// TIA Portal project "SERVO_2_AXIS" (V15.1)

(* hardware
DEVICE "S7-1200 station_1"  S7-1200 Station
   slot 0: "Rack_0"  S7-1200 Rack  Rack  V1.0
   slot 1: "PLC_1"  CPU 1214C DC/DC/DC  6ES7 214-1AG40-0XB0  V4.2
DEVICE "PC-System_1"  SIMATIC PC station
   slot 0: "SIMATIC PC station"  Rail  SIMATIC PC-Station  V1.0
      slot 125: "Stationmanager"  Station_Manager  V6.0.4
   slot 1: "HMI_RT_1"  WinCC RT Advanced  6AV2 104-0xxxx-xxxx  15.1.0.0
      slot 33792: "Host interface"  Host interface
   slot 2: "IE general_1"  IE General  IE_CP  V8.2.0
*)

// ===== PLC "PLC_1"  CPU 1214C DC/DC/DC =====

VAR_GLOBAL   // PLC tag table "Default tag table"
   "Axis_X_Pulse" AT %Q0.0 : Bool;
   "Axis_X_Direction" AT %Q0.1 : Bool;
   "Axis_Y_Pulse" AT %Q0.2 : Bool;
   "Axis_Y_Direction" AT %Q0.3 : Bool;
   "Tag_1" AT %M40.0 : Bool;
   "Set_Home_X" AT %M40.1 : Bool;
   "Thuận _X" AT %M40.2 : Bool;
   "Ngược_X" AT %M40.3 : Bool;
   "Speed_X" AT %MD10 : Real;
   "Enable_Y" AT %M50.0 : Bool;
   "Set_Home_Y" AT %M50.1 : Bool;
   "Thuận_Y" AT %M50.2 : Bool;
   "Ngược_Y" AT %M50.3 : Bool;
   "Speed_Y" AT %MD20 : Real;
   "Location_To_X" AT %MD14 : Real;
   "Start_X" AT %M40.4 : Bool;
   "Start_Y" AT %M50.4 : Bool;
   "Location_To_Y" AT %MD24 : Real;
   "Save_Location_X1" AT %M40.5 : Bool;
   "Save_Location_X2" AT %M40.6 : Bool;
   "Save_Location_X3" AT %M40.7 : Bool;
   "Save_Location_X4" AT %M41.0 : Bool;
   "Save_Location_X5" AT %M41.1 : Bool;
   "Save_Location_Y1" AT %M50.5 : Bool;
   "Save_Location_Y2" AT %M50.6 : Bool;
   "Save_Location_Y3" AT %M50.7 : Bool;
   "Save_Location_Y4" AT %M51.0 : Bool;
   "Save_Location_Y5" AT %M51.1 : Bool;
   "Input_location_X" AT %MW60 : Word;
   "Input_location_Y" AT %MW70 : Word;
   "System_Byte" AT %MB1 : Byte;
   "FirstScan" AT %M1.0 : Bool;
   "DiagStatusUpdate" AT %M1.1 : Bool;
   "AlwaysTRUE" AT %M1.2 : Bool;
   "AlwaysFALSE" AT %M1.3 : Bool;
   "X1" AT %M2.0 : Bool;
   "X2" AT %M2.1 : Bool;
   "X3" AT %M2.2 : Bool;
   "X4" AT %M2.3 : Bool;
   "X5" AT %M2.4 : Bool;
   "Y1" AT %M2.5 : Bool;
   "Y2" AT %M2.6 : Bool;
   "Y3" AT %M3.0 : Bool;
   "Y4" AT %M3.1 : Bool;
   "Y5" AT %M3.2 : Bool;
   "X1Y1" AT %M3.3 : Bool;
   "X1Y2" AT %M3.4 : Bool;
   "X1Y3" AT %M3.5 : Bool;
   "X1Y4" AT %M3.6 : Bool;
   "X1Y5" AT %M3.7 : Bool;
   "X2Y1" AT %M4.0 : Bool;
   "X2Y2" AT %M4.1 : Bool;
   "X2Y3" AT %M4.2 : Bool;
   "X2Y4" AT %M4.3 : Bool;
   "X2Y5" AT %M4.4 : Bool;
   "X3Y1" AT %M4.5 : Bool;
   "X3Y2" AT %M4.6 : Bool;
   "X3Y3" AT %M4.7 : Bool;
   "X3Y4" AT %M5.0 : Bool;
   "X3Y5" AT %M5.1 : Bool;
   "X4Y1" AT %M5.2 : Bool;
   "X4Y2" AT %M5.3 : Bool;
   "X4Y3" AT %M5.4 : Bool;
   "X4Y4" AT %M5.5 : Bool;
   "X4Y5" AT %M5.6 : Bool;
   "X5Y1" AT %M5.7 : Bool;
   "X5Y2" AT %M6.0 : Bool;
   "X5Y3" AT %M6.1 : Bool;
   "X5Y4" AT %M6.2 : Bool;
   "X5Y5" AT %M6.3 : Bool;
END_VAR

DATA_BLOCK "Location_X"   // DB3
{ S7_Optimized_Access := 'FALSE' }
VERSION : 0.1
   VAR
      Location_X : Array[1..5] of Real;
   END_VAR
BEGIN
END_DATA_BLOCK

DATA_BLOCK "Location_Y"   // DB4
{ S7_Optimized_Access := 'FALSE' }
VERSION : 0.1
   VAR
      Location_Y : Array[1..5] of Real;
   END_VAR
BEGIN
END_DATA_BLOCK

DATA_BLOCK "Axis_X"   // DB1, Motion_DB
{ S7_Optimized_Access := 'TRUE' }
AUTHOR : SIMATIC
FAMILY : BasicMC
NAME : TO_PosAx
VERSION : 6.0
// stored: InstanceOfName TO_PositioningAxis
"TO_PositioningAxis"
BEGIN
   // Axis.LengthUnitNormalized.Distance = 1013
   // Axis.DirectionOutputEnabledCU = TRUE
   // Axis.OnlinePtoModeCU = 16#0000_0002
   // Axis.SelectedChannel2EnumCU = %Q0.1
   // Axis.SelectedChannel1EnumCU = %Q0.0
   // Pulse.MinDeltaDeltaFrequencyCU = 0.004
   // Pulse.MaxDeltaDeltaFrequencyCU = 1.0E+10
   // Pulse.MinDeltaFrequencyCU = 0.005
   // Pulse.MaxDeltaFrequencyCU = 9.5E+9
   // Pulse.MinFrequencyCU = 1.0
   // Pulse.MaxFrequencyCU = 100000.0
   // Pulse.OutputSourceCU = 16#0000_0000
   // Axis.SelectPTO = 0
END_DATA_BLOCK

DATA_BLOCK "Axis_Y"   // DB2, Motion_DB
{ S7_Optimized_Access := 'TRUE' }
AUTHOR : SIMATIC
FAMILY : BasicMC
NAME : TO_PosAx
VERSION : 6.0
// stored: InstanceOfName TO_PositioningAxis
"TO_PositioningAxis"
BEGIN
   // Axis.LengthUnitNormalized.Distance = 1013
   // Axis.DirectionOutputEnabledCU = TRUE
   // Axis.OnlinePtoModeCU = 16#0000_0002
   // Axis.SelectedChannel2EnumCU = %Q0.3
   // Axis.SelectedChannel1EnumCU = %Q0.2
   // Pulse.MinDeltaDeltaFrequencyCU = 0.004
   // Pulse.MaxDeltaDeltaFrequencyCU = 1.0E+10
   // Pulse.MinDeltaFrequencyCU = 0.005
   // Pulse.MaxDeltaFrequencyCU = 9.5E+9
   // Pulse.MinFrequencyCU = 1.0
   // Pulse.MaxFrequencyCU = 100000.0
   // Pulse.OutputSourceCU = 16#0000_0000
   // Axis.SelectPTO = 1
   // Axis.OnlinePtoIndexCU = 1
END_DATA_BLOCK

FUNCTION "Power_X" : Void   // FC1, LAD
{ S7_Optimized_Access := 'TRUE' }
VERSION : 0.1
BEGIN

REGION Network 1
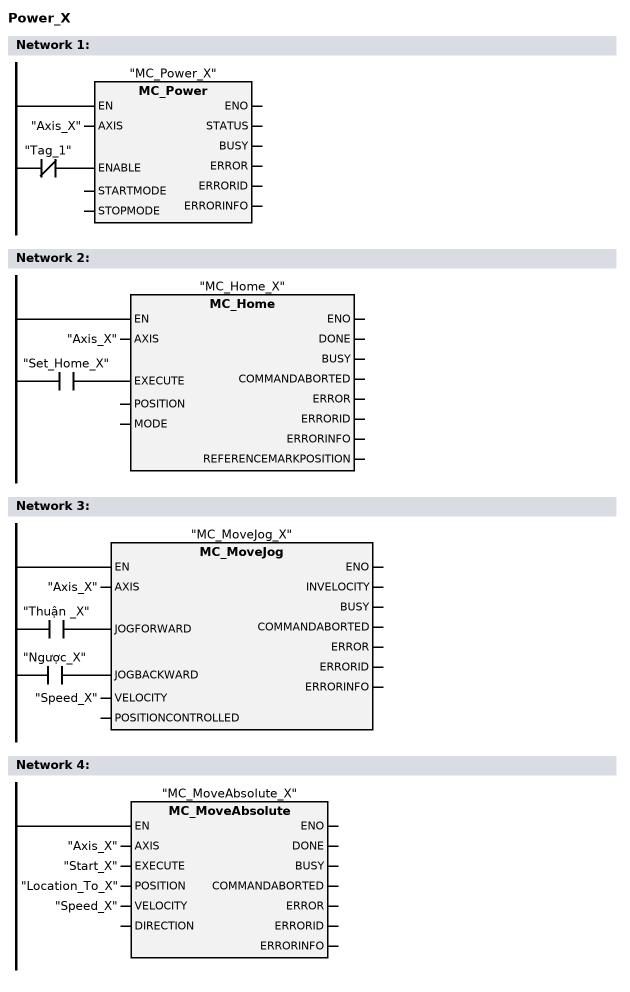
   "MC_Power_X"(Axis := "Axis_X", Enable := NOT "Tag_1");   // MC_Power
END_REGION

REGION Network 2
   "MC_Home_X"(Axis := "Axis_X", Execute := "Set_Home_X");   // MC_Home
END_REGION

REGION Network 3
   "MC_MoveJog_X"(Axis := "Axis_X", JogForward := "Thuận _X", JogBackward := "Ngược_X", Velocity := "Speed_X");   // MC_MoveJog
END_REGION

REGION Network 4
   "MC_MoveAbsolute_X"(Axis := "Axis_X",   // MC_MoveAbsolute
                       Execute := "Start_X",
                       Position := "Location_To_X",
                       Velocity := "Speed_X");
END_REGION
END_FUNCTION

FUNCTION "Power_Y" : Void   // FC2, LAD
{ S7_Optimized_Access := 'TRUE' }
VERSION : 0.1
BEGIN

REGION Network 1
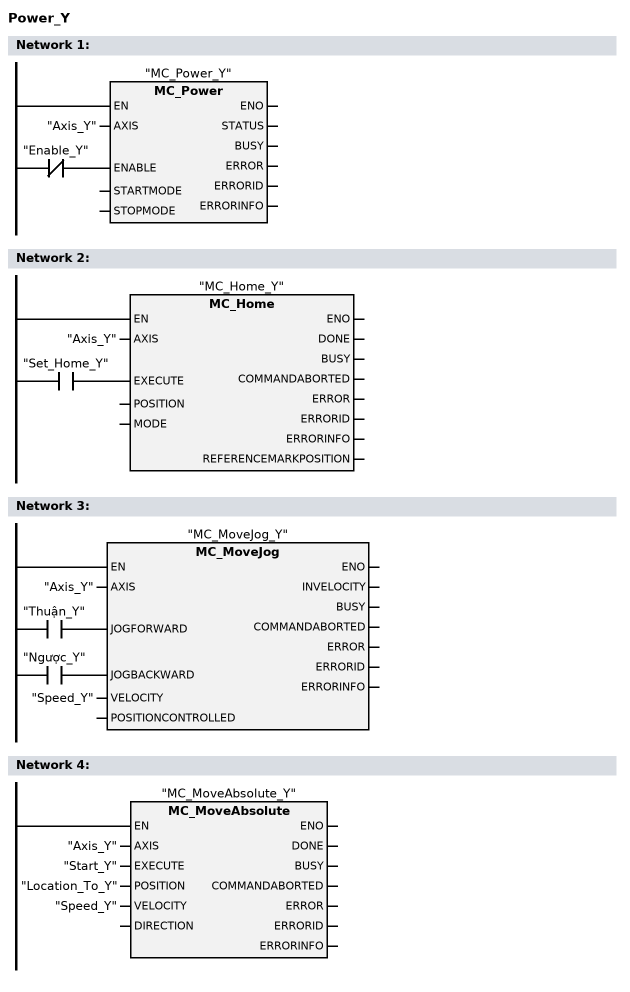
   "MC_Power_Y"(Axis := "Axis_Y", Enable := NOT "Enable_Y");   // MC_Power
END_REGION

REGION Network 2
   "MC_Home_Y"(Axis := "Axis_Y", Execute := "Set_Home_Y");   // MC_Home
END_REGION

REGION Network 3
   "MC_MoveJog_Y"(Axis := "Axis_Y", JogForward := "Thuận_Y", JogBackward := "Ngược_Y", Velocity := "Speed_Y");   // MC_MoveJog
END_REGION

REGION Network 4
   "MC_MoveAbsolute_Y"(Axis := "Axis_Y",   // MC_MoveAbsolute
                       Execute := "Start_Y",
                       Position := "Location_To_Y",
                       Velocity := "Speed_Y");
END_REGION
END_FUNCTION

FUNCTION "Save_Location_X" : Void   // FC3, LAD
{ S7_Optimized_Access := 'TRUE' }
VERSION : 0.1
BEGIN

REGION Network 1
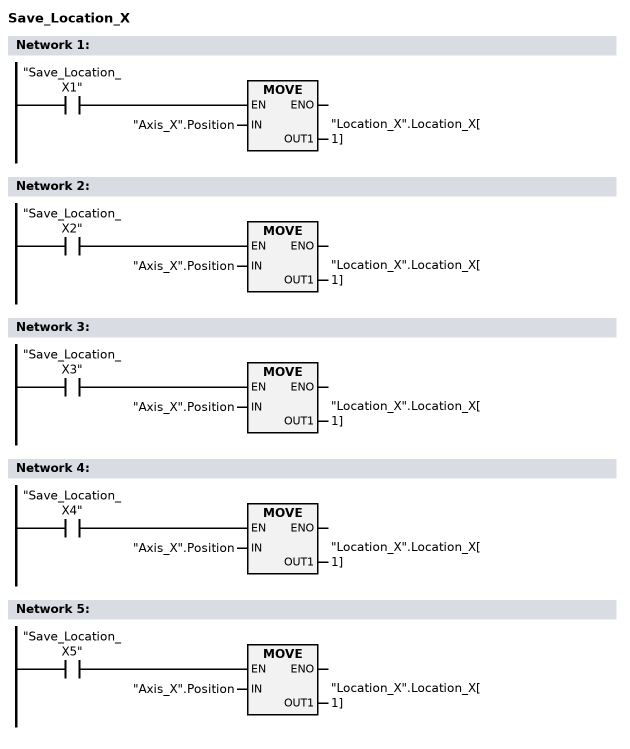
   RUNG wire#powerrail
      Contact( "Save_Location_X1" )
      Move(in := "Axis_X".Position, out1 => "Location_X".Location_X[1])
   END_RUNG
   // the same network as SCL:
   IF "Save_Location_X1" THEN "Location_X".Location_X[1] := "Axis_X".Position; END_IF;
END_REGION

REGION Network 2
   RUNG wire#powerrail
      Contact( "Save_Location_X2" )
      Move(in := "Axis_X".Position, out1 => "Location_X".Location_X[1])
   END_RUNG
   // the same network as SCL:
   IF "Save_Location_X2" THEN "Location_X".Location_X[1] := "Axis_X".Position; END_IF;
END_REGION

REGION Network 3
   RUNG wire#powerrail
      Contact( "Save_Location_X3" )
      Move(in := "Axis_X".Position, out1 => "Location_X".Location_X[1])
   END_RUNG
   // the same network as SCL:
   IF "Save_Location_X3" THEN "Location_X".Location_X[1] := "Axis_X".Position; END_IF;
END_REGION

REGION Network 4
   RUNG wire#powerrail
      Contact( "Save_Location_X4" )
      Move(in := "Axis_X".Position, out1 => "Location_X".Location_X[1])
   END_RUNG
   // the same network as SCL:
   IF "Save_Location_X4" THEN "Location_X".Location_X[1] := "Axis_X".Position; END_IF;
END_REGION

REGION Network 5
   RUNG wire#powerrail
      Contact( "Save_Location_X5" )
      Move(in := "Axis_X".Position, out1 => "Location_X".Location_X[1])
   END_RUNG
   // the same network as SCL:
   IF "Save_Location_X5" THEN "Location_X".Location_X[1] := "Axis_X".Position; END_IF;
END_REGION
END_FUNCTION

FUNCTION "Save_Location_Y" : Void   // FC4, LAD
{ S7_Optimized_Access := 'TRUE' }
VERSION : 0.1
BEGIN

REGION Network 1
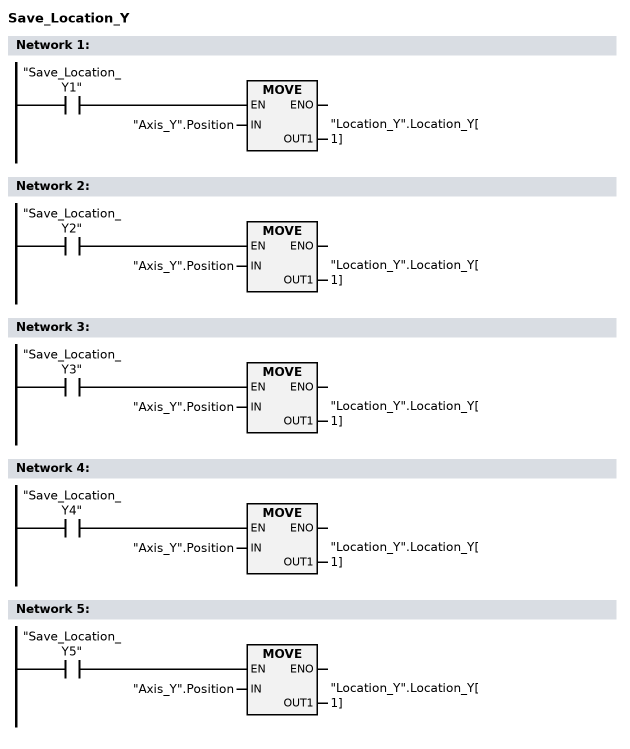
   RUNG wire#powerrail
      Contact( "Save_Location_Y1" )
      Move(in := "Axis_Y".Position, out1 => "Location_Y".Location_Y[1])
   END_RUNG
   // the same network as SCL:
   IF "Save_Location_Y1" THEN "Location_Y".Location_Y[1] := "Axis_Y".Position; END_IF;
END_REGION

REGION Network 2
   RUNG wire#powerrail
      Contact( "Save_Location_Y2" )
      Move(in := "Axis_Y".Position, out1 => "Location_Y".Location_Y[1])
   END_RUNG
   // the same network as SCL:
   IF "Save_Location_Y2" THEN "Location_Y".Location_Y[1] := "Axis_Y".Position; END_IF;
END_REGION

REGION Network 3
   RUNG wire#powerrail
      Contact( "Save_Location_Y3" )
      Move(in := "Axis_Y".Position, out1 => "Location_Y".Location_Y[1])
   END_RUNG
   // the same network as SCL:
   IF "Save_Location_Y3" THEN "Location_Y".Location_Y[1] := "Axis_Y".Position; END_IF;
END_REGION

REGION Network 4
   RUNG wire#powerrail
      Contact( "Save_Location_Y4" )
      Move(in := "Axis_Y".Position, out1 => "Location_Y".Location_Y[1])
   END_RUNG
   // the same network as SCL:
   IF "Save_Location_Y4" THEN "Location_Y".Location_Y[1] := "Axis_Y".Position; END_IF;
END_REGION

REGION Network 5
   RUNG wire#powerrail
      Contact( "Save_Location_Y5" )
      Move(in := "Axis_Y".Position, out1 => "Location_Y".Location_Y[1])
   END_RUNG
   // the same network as SCL:
   IF "Save_Location_Y5" THEN "Location_Y".Location_Y[1] := "Axis_Y".Position; END_IF;
END_REGION
END_FUNCTION

FUNCTION "Call_Location_X" : Void   // FC5, LAD
{ S7_Optimized_Access := 'TRUE' }
VERSION : 0.1
BEGIN

REGION Network 1
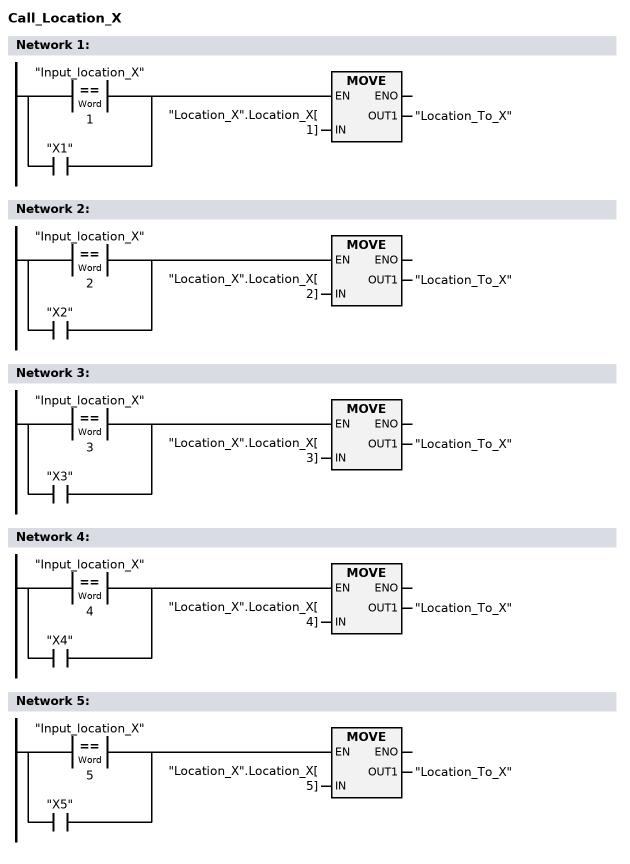
   RUNG wire#powerrail
      { S7_Templates := "SrcType := Word" } EQ_Contact(in1 := "Input_location_X", in2 := 1)
      wire#w1
      Move(in := "Location_X".Location_X[1], out1 => "Location_To_X")
   END_RUNG
   RUNG wire#powerrail
      Contact( "X1" )
   END_RUNG wire#w1
   // the same network as SCL:
   IF ("Input_location_X" = 1) OR "X1" THEN "Location_To_X" := "Location_X".Location_X[1]; END_IF;
END_REGION

REGION Network 2
   RUNG wire#powerrail
      { S7_Templates := "SrcType := Word" } EQ_Contact(in1 := "Input_location_X", in2 := 2)
      wire#w1
      Move(in := "Location_X".Location_X[2], out1 => "Location_To_X")
   END_RUNG
   RUNG wire#powerrail
      Contact( "X2" )
   END_RUNG wire#w1
   // the same network as SCL:
   IF ("Input_location_X" = 2) OR "X2" THEN "Location_To_X" := "Location_X".Location_X[2]; END_IF;
END_REGION

REGION Network 3
   RUNG wire#powerrail
      { S7_Templates := "SrcType := Word" } EQ_Contact(in1 := "Input_location_X", in2 := 3)
      wire#w1
      Move(in := "Location_X".Location_X[3], out1 => "Location_To_X")
   END_RUNG
   RUNG wire#powerrail
      Contact( "X3" )
   END_RUNG wire#w1
   // the same network as SCL:
   IF ("Input_location_X" = 3) OR "X3" THEN "Location_To_X" := "Location_X".Location_X[3]; END_IF;
END_REGION

REGION Network 4
   RUNG wire#powerrail
      { S7_Templates := "SrcType := Word" } EQ_Contact(in1 := "Input_location_X", in2 := 4)
      wire#w1
      Move(in := "Location_X".Location_X[4], out1 => "Location_To_X")
   END_RUNG
   RUNG wire#powerrail
      Contact( "X4" )
   END_RUNG wire#w1
   // the same network as SCL:
   IF ("Input_location_X" = 4) OR "X4" THEN "Location_To_X" := "Location_X".Location_X[4]; END_IF;
END_REGION

REGION Network 5
   RUNG wire#powerrail
      { S7_Templates := "SrcType := Word" } EQ_Contact(in1 := "Input_location_X", in2 := 5)
      wire#w1
      Move(in := "Location_X".Location_X[5], out1 => "Location_To_X")
   END_RUNG
   RUNG wire#powerrail
      Contact( "X5" )
   END_RUNG wire#w1
   // the same network as SCL:
   IF ("Input_location_X" = 5) OR "X5" THEN "Location_To_X" := "Location_X".Location_X[5]; END_IF;
END_REGION
END_FUNCTION

FUNCTION "Call_Location_Y" : Void   // FC6, LAD
{ S7_Optimized_Access := 'TRUE' }
VERSION : 0.1
BEGIN

REGION Network 1
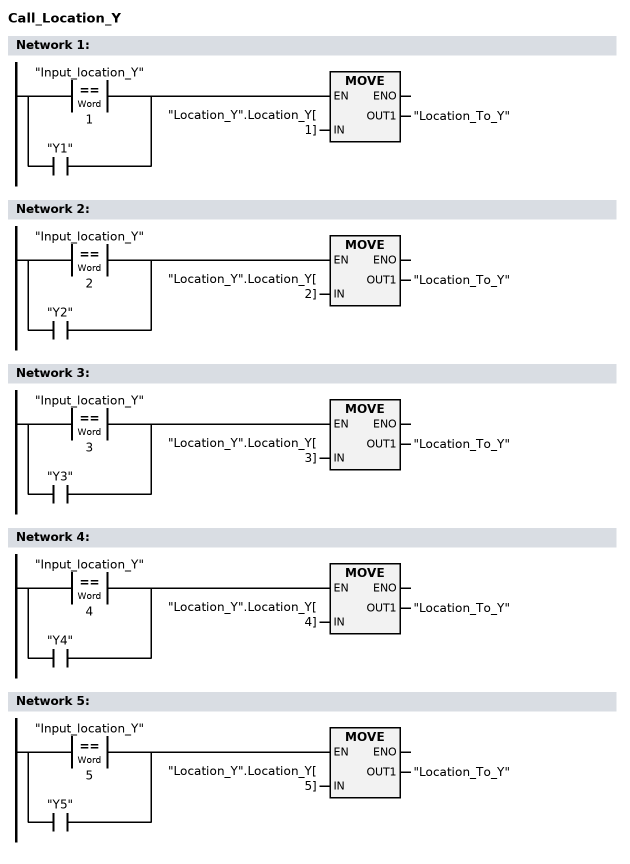
   RUNG wire#powerrail
      { S7_Templates := "SrcType := Word" } EQ_Contact(in1 := "Input_location_Y", in2 := 1)
      wire#w1
      Move(in := "Location_Y".Location_Y[1], out1 => "Location_To_Y")
   END_RUNG
   RUNG wire#powerrail
      Contact( "Y1" )
   END_RUNG wire#w1
   // the same network as SCL:
   IF ("Input_location_Y" = 1) OR "Y1" THEN "Location_To_Y" := "Location_Y".Location_Y[1]; END_IF;
END_REGION

REGION Network 2
   RUNG wire#powerrail
      { S7_Templates := "SrcType := Word" } EQ_Contact(in1 := "Input_location_Y", in2 := 2)
      wire#w1
      Move(in := "Location_Y".Location_Y[2], out1 => "Location_To_Y")
   END_RUNG
   RUNG wire#powerrail
      Contact( "Y2" )
   END_RUNG wire#w1
   // the same network as SCL:
   IF ("Input_location_Y" = 2) OR "Y2" THEN "Location_To_Y" := "Location_Y".Location_Y[2]; END_IF;
END_REGION

REGION Network 3
   RUNG wire#powerrail
      { S7_Templates := "SrcType := Word" } EQ_Contact(in1 := "Input_location_Y", in2 := 3)
      wire#w1
      Move(in := "Location_Y".Location_Y[3], out1 => "Location_To_Y")
   END_RUNG
   RUNG wire#powerrail
      Contact( "Y3" )
   END_RUNG wire#w1
   // the same network as SCL:
   IF ("Input_location_Y" = 3) OR "Y3" THEN "Location_To_Y" := "Location_Y".Location_Y[3]; END_IF;
END_REGION

REGION Network 4
   RUNG wire#powerrail
      { S7_Templates := "SrcType := Word" } EQ_Contact(in1 := "Input_location_Y", in2 := 4)
      wire#w1
      Move(in := "Location_Y".Location_Y[4], out1 => "Location_To_Y")
   END_RUNG
   RUNG wire#powerrail
      Contact( "Y4" )
   END_RUNG wire#w1
   // the same network as SCL:
   IF ("Input_location_Y" = 4) OR "Y4" THEN "Location_To_Y" := "Location_Y".Location_Y[4]; END_IF;
END_REGION

REGION Network 5
   RUNG wire#powerrail
      { S7_Templates := "SrcType := Word" } EQ_Contact(in1 := "Input_location_Y", in2 := 5)
      wire#w1
      Move(in := "Location_Y".Location_Y[5], out1 => "Location_To_Y")
   END_RUNG
   RUNG wire#powerrail
      Contact( "Y5" )
   END_RUNG wire#w1
   // the same network as SCL:
   IF ("Input_location_Y" = 5) OR "Y5" THEN "Location_To_Y" := "Location_Y".Location_Y[5]; END_IF;
END_REGION
END_FUNCTION

FUNCTION "XY" : Void   // FC7, LAD
{ S7_Optimized_Access := 'TRUE' }
VERSION : 0.1
BEGIN

REGION Network 1
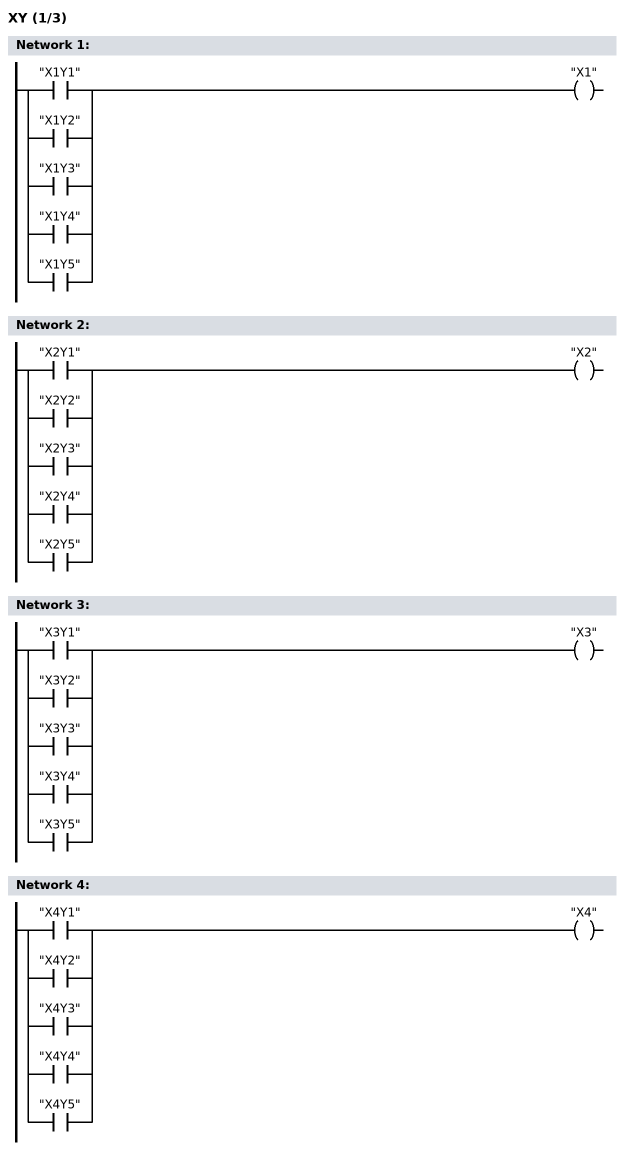
   RUNG wire#powerrail
      Contact( "X1Y1" )
      wire#w1
      Coil( "X1" )
   END_RUNG
   RUNG wire#powerrail
      Contact( "X1Y2" )
   END_RUNG wire#w1
   RUNG wire#powerrail
      Contact( "X1Y3" )
   END_RUNG wire#w1
   RUNG wire#powerrail
      Contact( "X1Y4" )
   END_RUNG wire#w1
   RUNG wire#powerrail
      Contact( "X1Y5" )
   END_RUNG wire#w1
   // the same network as SCL:
   "X1" := "X1Y1" OR "X1Y2" OR "X1Y3" OR "X1Y4" OR "X1Y5";
END_REGION

REGION Network 2
   RUNG wire#powerrail
      Contact( "X2Y1" )
      wire#w1
      Coil( "X2" )
   END_RUNG
   RUNG wire#powerrail
      Contact( "X2Y2" )
   END_RUNG wire#w1
   RUNG wire#powerrail
      Contact( "X2Y3" )
   END_RUNG wire#w1
   RUNG wire#powerrail
      Contact( "X2Y4" )
   END_RUNG wire#w1
   RUNG wire#powerrail
      Contact( "X2Y5" )
   END_RUNG wire#w1
   // the same network as SCL:
   "X2" := "X2Y1" OR "X2Y2" OR "X2Y3" OR "X2Y4" OR "X2Y5";
END_REGION

REGION Network 3
   RUNG wire#powerrail
      Contact( "X3Y1" )
      wire#w1
      Coil( "X3" )
   END_RUNG
   RUNG wire#powerrail
      Contact( "X3Y2" )
   END_RUNG wire#w1
   RUNG wire#powerrail
      Contact( "X3Y3" )
   END_RUNG wire#w1
   RUNG wire#powerrail
      Contact( "X3Y4" )
   END_RUNG wire#w1
   RUNG wire#powerrail
      Contact( "X3Y5" )
   END_RUNG wire#w1
   // the same network as SCL:
   "X3" := "X3Y1" OR "X3Y2" OR "X3Y3" OR "X3Y4" OR "X3Y5";
END_REGION

REGION Network 4
   RUNG wire#powerrail
      Contact( "X4Y1" )
      wire#w1
      Coil( "X4" )
   END_RUNG
   RUNG wire#powerrail
      Contact( "X4Y2" )
   END_RUNG wire#w1
   RUNG wire#powerrail
      Contact( "X4Y3" )
   END_RUNG wire#w1
   RUNG wire#powerrail
      Contact( "X4Y4" )
   END_RUNG wire#w1
   RUNG wire#powerrail
      Contact( "X4Y5" )
   END_RUNG wire#w1
   // the same network as SCL:
   "X4" := "X4Y1" OR "X4Y2" OR "X4Y3" OR "X4Y4" OR "X4Y5";
END_REGION

REGION Network 5
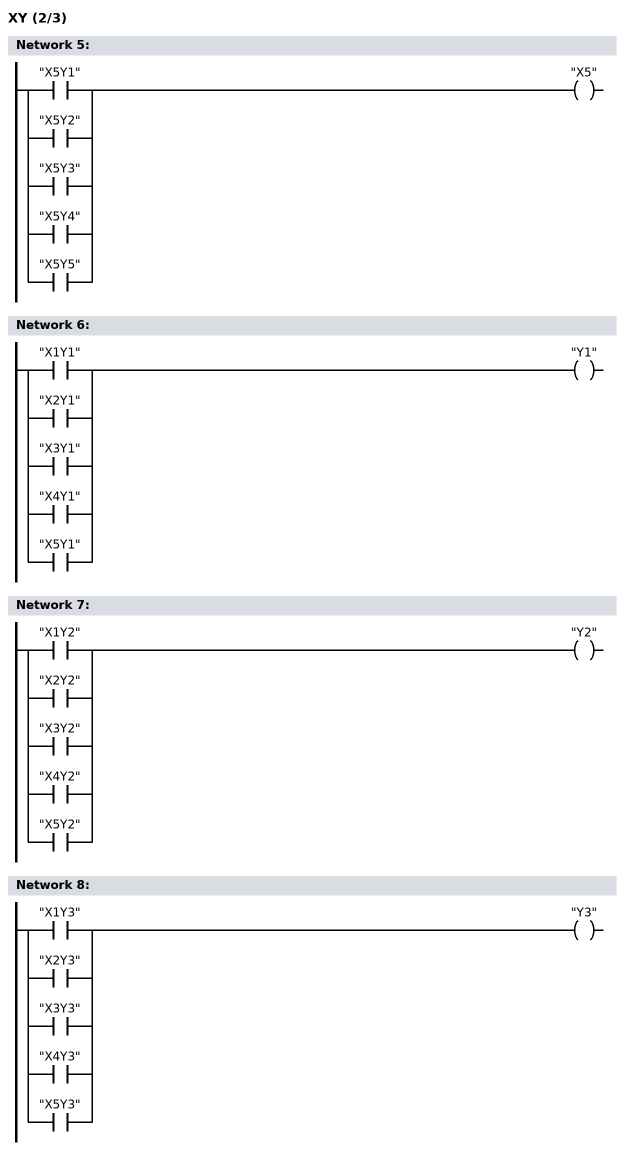
   RUNG wire#powerrail
      Contact( "X5Y1" )
      wire#w1
      Coil( "X5" )
   END_RUNG
   RUNG wire#powerrail
      Contact( "X5Y2" )
   END_RUNG wire#w1
   RUNG wire#powerrail
      Contact( "X5Y3" )
   END_RUNG wire#w1
   RUNG wire#powerrail
      Contact( "X5Y4" )
   END_RUNG wire#w1
   RUNG wire#powerrail
      Contact( "X5Y5" )
   END_RUNG wire#w1
   // the same network as SCL:
   "X5" := "X5Y1" OR "X5Y2" OR "X5Y3" OR "X5Y4" OR "X5Y5";
END_REGION

REGION Network 6
   RUNG wire#powerrail
      Contact( "X1Y1" )
      wire#w1
      Coil( "Y1" )
   END_RUNG
   RUNG wire#powerrail
      Contact( "X2Y1" )
   END_RUNG wire#w1
   RUNG wire#powerrail
      Contact( "X3Y1" )
   END_RUNG wire#w1
   RUNG wire#powerrail
      Contact( "X4Y1" )
   END_RUNG wire#w1
   RUNG wire#powerrail
      Contact( "X5Y1" )
   END_RUNG wire#w1
   // the same network as SCL:
   "Y1" := "X1Y1" OR "X2Y1" OR "X3Y1" OR "X4Y1" OR "X5Y1";
END_REGION

REGION Network 7
   RUNG wire#powerrail
      Contact( "X1Y2" )
      wire#w1
      Coil( "Y2" )
   END_RUNG
   RUNG wire#powerrail
      Contact( "X2Y2" )
   END_RUNG wire#w1
   RUNG wire#powerrail
      Contact( "X3Y2" )
   END_RUNG wire#w1
   RUNG wire#powerrail
      Contact( "X4Y2" )
   END_RUNG wire#w1
   RUNG wire#powerrail
      Contact( "X5Y2" )
   END_RUNG wire#w1
   // the same network as SCL:
   "Y2" := "X1Y2" OR "X2Y2" OR "X3Y2" OR "X4Y2" OR "X5Y2";
END_REGION

REGION Network 8
   RUNG wire#powerrail
      Contact( "X1Y3" )
      wire#w1
      Coil( "Y3" )
   END_RUNG
   RUNG wire#powerrail
      Contact( "X2Y3" )
   END_RUNG wire#w1
   RUNG wire#powerrail
      Contact( "X3Y3" )
   END_RUNG wire#w1
   RUNG wire#powerrail
      Contact( "X4Y3" )
   END_RUNG wire#w1
   RUNG wire#powerrail
      Contact( "X5Y3" )
   END_RUNG wire#w1
   // the same network as SCL:
   "Y3" := "X1Y3" OR "X2Y3" OR "X3Y3" OR "X4Y3" OR "X5Y3";
END_REGION

REGION Network 9
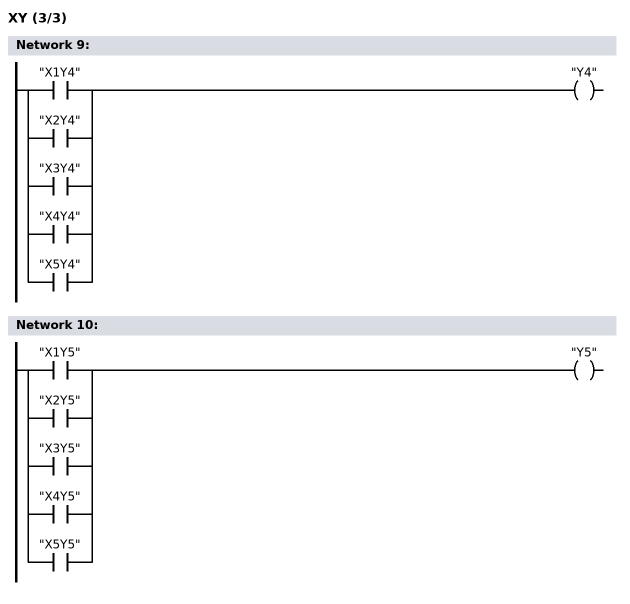
   RUNG wire#powerrail
      Contact( "X1Y4" )
      wire#w1
      Coil( "Y4" )
   END_RUNG
   RUNG wire#powerrail
      Contact( "X2Y4" )
   END_RUNG wire#w1
   RUNG wire#powerrail
      Contact( "X3Y4" )
   END_RUNG wire#w1
   RUNG wire#powerrail
      Contact( "X4Y4" )
   END_RUNG wire#w1
   RUNG wire#powerrail
      Contact( "X5Y4" )
   END_RUNG wire#w1
   // the same network as SCL:
   "Y4" := "X1Y4" OR "X2Y4" OR "X3Y4" OR "X4Y4" OR "X5Y4";
END_REGION

REGION Network 10
   RUNG wire#powerrail
      Contact( "X1Y5" )
      wire#w1
      Coil( "Y5" )
   END_RUNG
   RUNG wire#powerrail
      Contact( "X2Y5" )
   END_RUNG wire#w1
   RUNG wire#powerrail
      Contact( "X3Y5" )
   END_RUNG wire#w1
   RUNG wire#powerrail
      Contact( "X4Y5" )
   END_RUNG wire#w1
   RUNG wire#powerrail
      Contact( "X5Y5" )
   END_RUNG wire#w1
   // the same network as SCL:
   "Y5" := "X1Y5" OR "X2Y5" OR "X3Y5" OR "X4Y5" OR "X5Y5";
END_REGION
END_FUNCTION

ORGANIZATION_BLOCK "Main"   // OB1, LAD, ProgramCycle
TITLE = "Main Program Sweep (Cycle)"
{ S7_Optimized_Access := 'TRUE' }
VERSION : 0.1
   VAR_INPUT
      Initial_Call : Bool;   // Initial call of this OB
      Remanence : Bool;   // =True, if remanent data are available
   END_VAR
   VAR_TEMP   // added for the SCL form of the ladder/FBD networks
      _w1 : Bool;
   END_VAR
BEGIN

REGION Network 1
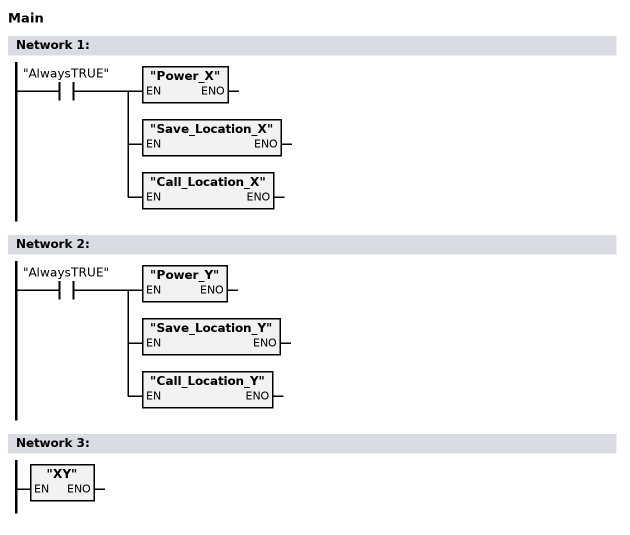
   RUNG wire#powerrail
      Contact( "AlwaysTRUE" )
      wire#w1
      "Power_X"()
   END_RUNG
   RUNG wire#w1
      "Save_Location_X"()
   END_RUNG
   RUNG wire#w1
      "Call_Location_X"()
   END_RUNG
   // the same network as SCL:
   #_w1 := "AlwaysTRUE";
   IF #_w1 THEN
       "Power_X"();
       "Save_Location_X"();
       "Call_Location_X"();
   END_IF;
END_REGION

REGION Network 2
   RUNG wire#powerrail
      Contact( "AlwaysTRUE" )
      wire#w1
      "Power_Y"()
   END_RUNG
   RUNG wire#w1
      "Save_Location_Y"()
   END_RUNG
   RUNG wire#w1
      "Call_Location_Y"()
   END_RUNG
   // the same network as SCL:
   #_w1 := "AlwaysTRUE";
   IF #_w1 THEN
       "Power_Y"();
       "Save_Location_Y"();
       "Call_Location_Y"();
   END_IF;
END_REGION

REGION Network 3
   RUNG wire#powerrail
      "XY"()
   END_RUNG
   // the same network as SCL:
   "XY"();
END_REGION
END_ORGANIZATION_BLOCK

(* ===== HMI "HMI_RT_1" =====
system functions are stored by id; their names below are inferred from use
connection "HMI_Connection_1": ETHERNET, S7_1200_OMS

HMI tags "Default tag table"
   "X1Y1" : Bool = PLC X1Y1 AT %M3.3, 100 ms
   "X2Y1" : Bool = PLC X2Y1 AT %M4.0, 100 ms
   "X1Y2" : Bool = PLC X1Y2 AT %M3.4, 100 ms
   "X1Y3" : Bool = PLC X1Y3 AT %M3.5, 100 ms
   "X1Y4" : Bool = PLC X1Y4 AT %M3.6, 100 ms
   "X1Y5" : Bool = PLC X1Y5 AT %M3.7, 100 ms
   "X2Y2" : Bool = PLC X2Y2 AT %M4.1, 100 ms
   "X2Y3" : Bool = PLC X2Y3 AT %M4.2, 100 ms
   "X2Y4" : Bool = PLC X2Y4 AT %M4.3, 100 ms
   "X2Y5" : Bool = PLC X2Y5 AT %M4.4, 100 ms
   "X3Y1" : Bool = PLC X3Y1 AT %M4.5, 100 ms
   "X3Y2" : Bool = PLC X3Y2 AT %M4.6, 100 ms
   "X3Y3" : Bool = PLC X3Y3 AT %M4.7, 100 ms
   "X3Y4" : Bool = PLC X3Y4 AT %M5.0, 100 ms
   "X3Y5" : Bool = PLC X3Y5 AT %M5.1, 100 ms
   "X4Y1" : Bool = PLC X4Y1 AT %M5.2, 100 ms
   "X4Y2" : Bool = PLC X4Y2 AT %M5.3, 100 ms
   "X4Y3" : Bool = PLC X4Y3 AT %M5.4, 100 ms
   "X4Y4" : Bool = PLC X4Y4 AT %M5.5, 100 ms
   "X4Y5" : Bool = PLC X4Y5 AT %M5.6, 100 ms
   "X5Y1" : Bool = PLC X5Y1 AT %M5.7, 100 ms
   "X5Y2" : Bool = PLC X5Y2 AT %M6.0, 100 ms
   "X5Y3" : Bool = PLC X5Y3 AT %M6.1, 100 ms
   "X5Y4" : Bool = PLC X5Y4 AT %M6.2, 100 ms
   "X5Y5" : Bool = PLC X5Y5 AT %M6.3, 100 ms
   "X1" : Bool = PLC X1 AT %M2.0, 100 ms
   "X2" : Bool = PLC X2 AT %M2.1, 100 ms
   "X3" : Bool = PLC X3 AT %M2.2, 100 ms
   "X4" : Bool = PLC X4 AT %M2.3, 100 ms
   "X5" : Bool = PLC X5 AT %M2.4, 100 ms
   "Y1" : Bool = PLC Y1 AT %M2.5, 100 ms
   "Y2" : Bool = PLC Y2 AT %M2.6, 100 ms
   "Y3" : Bool = PLC Y3 AT %M3.0, 100 ms
   "Y4" : Bool = PLC Y4 AT %M3.1, 100 ms
   "Y5" : Bool = PLC Y5 AT %M3.2, 100 ms

screen "Screen_1" 1024x768
   Button "Button_1" at 68,227 size 69x32; TextOff 'X1Y1'
      on Press: SetBit("X1Y1")
      on Release: ResetBit("X1Y1")
   Button "Button_2" at 68,260 size 69x32; TextOff 'X1Y2'
      on Press: SetBit("X1Y2")
      on Release: ResetBit("X1Y2")
   Button "Button_3" at 68,293 size 69x32; TextOff 'X1Y3'
      on Press: SetBit("X1Y3")
      on Release: ResetBit("X1Y3")
   Button "Button_4" at 68,325 size 69x32; TextOff 'X1Y4'
      on Press: SetBit("X1Y4")
      on Release: ResetBit("X1Y4")
   Button "Button_5" at 68,358 size 69x32; TextOff 'X1Y5'
      on Press: SetBit("X1Y5")
      on Release: ResetBit("X1Y5")
   Button "Button_6" at 138,227 size 69x32; TextOff 'X2Y1'
      on Press: SetBit("X2Y1")
      on Release: ResetBit("X2Y1")
   Button "Button_7" at 138,260 size 69x32; TextOff 'X2Y2'
      on Press: SetBit("X2Y2")
      on Release: ResetBit("X2Y2")
   Button "Button_8" at 138,293 size 69x32; TextOff 'X2Y3'
      on Press: SetBit("X2Y3")
      on Release: ResetBit("X2Y3")
   Button "Button_9" at 138,325 size 69x32; TextOff 'X2Y4'
      on Press: SetBit("X2Y4")
      on Release: ResetBit("X2Y4")
   Button "Button_10" at 138,358 size 69x32; TextOff 'X2Y5'
      on Release: ResetBit("X2Y5")
      on Press: SetBit("X2Y5")
   Button "Button_11" at 208,227 size 69x32; TextOff 'X3Y1'
      on Release: ResetBit("X3Y1")
      on Press: SetBit("X3Y1")
   Button "Button_12" at 208,260 size 69x32; TextOff 'X3Y2'
      on Press: SetBit("X3Y2")
      on Release: ResetBit("X3Y2")
   Button "Button_13" at 208,293 size 69x32; TextOff 'X3Y3'
      on Press: SetBit("X3Y3")
      on Release: ResetBit("X3Y3")
   Button "Button_14" at 208,325 size 69x32; TextOff 'X3Y4'
      on Press: SetBit("X3Y4")
      on Release: ResetBit("X3Y4")
   Button "Button_15" at 208,358 size 69x32; TextOff 'X3Y5'
      on Press: SetBit("X3Y5")
      on Release: ResetBit("X3Y5")
   Button "Button_16" at 278,227 size 69x32; TextOff 'X4Y1'
      on Press: SetBit("X4Y1")
      on Release: ResetBit("X4Y1")
   Button "Button_17" at 278,260 size 69x32; TextOff 'X4Y2'
      on Press: SetBit("X4Y2")
      on Release: ResetBit("X4Y2")
   Button "Button_18" at 278,293 size 69x32; TextOff 'X4Y3'
      on Press: SetBit("X4Y3")
      on Release: ResetBit("X4Y3")
   Button "Button_19" at 278,325 size 69x32; TextOff 'X4Y4'
      on Press: SetBit("X4Y4")
      on Release: ResetBit("X4Y4")
   Button "Button_20" at 278,358 size 69x32; TextOff 'X4Y5'
      on Press: SetBit("X4Y5")
      on Release: ResetBit("X4Y5")
   Button "Button_21" at 348,227 size 69x32; TextOff 'X5Y1'
      on Press: SetBit("X5Y1")
      on Release: ResetBit("X5Y1")
   Button "Button_22" at 348,260 size 69x32; TextOff 'X5Y2'
      on Press: SetBit("X5Y2")
      on Release: ResetBit("X5Y2")
   Button "Button_23" at 348,293 size 69x32; TextOff 'X5Y3'
      on Press: SetBit("X5Y3")
      on Release: ResetBit("X5Y3")
   Button "Button_24" at 348,325 size 69x32; TextOff 'X5Y4'
      on Press: SetBit("X5Y4")
      on Release: ResetBit("X5Y4")
   Button "Button_25" at 348,358 size 69x32; TextOff 'X5Y5'
      on Press: SetBit("X5Y5")
      on Release: ResetBit("X5Y5")
   Circle "Circle_1" at 94,103 size 48x48
      Appearance <- "X1"
   Circle "Circle_2" at 94,162 size 48x48
      Appearance <- "Y1"
   Circle "Circle_3" at 156,103 size 48x48
      Appearance <- "X2"
   Circle "Circle_4" at 156,162 size 48x48
      Appearance <- "Y2"
   Circle "Circle_5" at 218,103 size 48x48
      Appearance <- "X3"
   Circle "Circle_6" at 218,162 size 48x48
      Appearance <- "Y3"
   Circle "Circle_7" at 280,103 size 48x48
      Appearance <- "X4"
   Circle "Circle_8" at 280,162 size 48x48
      Appearance <- "Y4"
   Circle "Circle_9" at 343,103 size 48x48
      Appearance <- "X5"
   Circle "Circle_10" at 343,162 size 48x48
      Appearance <- "Y5"
*)